FUNCTION_BLOCK UT_AuxiliaryInputMapping_Type_13_QuadratAnalog_Ret50perc (* Two quadrature mounted analog returns to centre position at 50% *)
  (* Standard: ISO 11783-6; Classification: AUX – ISO 11783-6; Function: All Inputs; Type: UT according to ISO 11783-6; Description: - Type 13 QuadratAnalog_Ret50perc Two quadrature mounted analog returns to centre position at 50% Applicable AUX-N only * maps to IW IW - Input WORD (16 Bit) *)
  (* Version 1.0, 2018-12-05, Jose Cabral *)
  (* Version 1.1, 2022-08-04, Franz Hoepfinger, HR Agrartechnik GmbH *)
  (* Version 1.2, 2023-01-05, Franz Hoepfinger, HR Agrartechnik GmbH *)
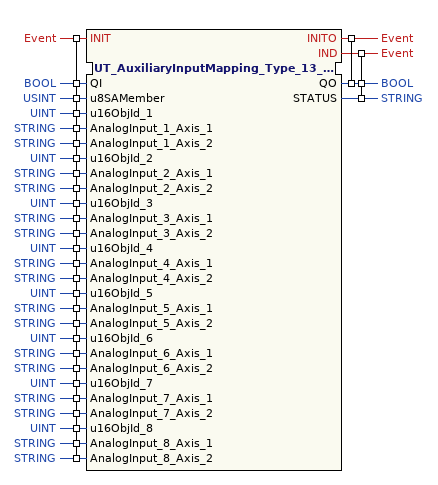
  EVENT_INPUT
    INIT WITH QI, u8SAMember, u16ObjId_1, AnalogInput_1_Axis_1, AnalogInput_1_Axis_2, u16ObjId_2, AnalogInput_2_Axis_1, AnalogInput_2_Axis_2, u16ObjId_3, AnalogInput_3_Axis_1, AnalogInput_3_Axis_2, u16ObjId_4, AnalogInput_4_Axis_1, AnalogInput_4_Axis_2, u16ObjId_5, AnalogInput_5_Axis_1, AnalogInput_5_Axis_2, u16ObjId_6, AnalogInput_6_Axis_1, AnalogInput_6_Axis_2, u16ObjId_7, AnalogInput_7_Axis_1, AnalogInput_7_Axis_2, u16ObjId_8, AnalogInput_8_Axis_1, AnalogInput_8_Axis_2; (* Service Initialization *)
  END_EVENT
  EVENT_OUTPUT
    INITO WITH QO; (* Initialization Confirm *)
    IND WITH QO, STATUS; (* Indication from Resource *)
  END_EVENT
  VAR_INPUT
    QI : BOOL; (* Event Input Qualifier *)
    u8SAMember : USINT := GLOBAL; (* Dummy !, set to GLOBAL if in doubt. OFF deactivates FB. *)
    u16ObjId_1 : UINT; (* Object ID of Input 1 *)
    AnalogInput_1_Axis_1 : STRING; (* Identifier for Input 1 Axis #1 *)
    AnalogInput_1_Axis_2 : STRING; (* Identifier for Input 1 Axis #2 *)
    u16ObjId_2 : UINT; (* Object ID of Input 2 *)
    AnalogInput_2_Axis_1 : STRING; (* Identifier for Input 2 Axis #1 *)
    AnalogInput_2_Axis_2 : STRING; (* Identifier for Input 2 Axis #2 *)
    u16ObjId_3 : UINT; (* Object ID of Input 3 *)
    AnalogInput_3_Axis_1 : STRING; (* Identifier for Input 3 Axis #1 *)
    AnalogInput_3_Axis_2 : STRING; (* Identifier for Input 3 Axis #2 *)
    u16ObjId_4 : UINT; (* Object ID of Input 4 *)
    AnalogInput_4_Axis_1 : STRING; (* Identifier for Input 4 Axis #1 *)
    AnalogInput_4_Axis_2 : STRING; (* Identifier for Input 4 Axis #2 *)
    u16ObjId_5 : UINT; (* Object ID of Input 5 *)
    AnalogInput_5_Axis_1 : STRING; (* Identifier for Input 5 Axis #1 *)
    AnalogInput_5_Axis_2 : STRING; (* Identifier for Input 5 Axis #2 *)
    u16ObjId_6 : UINT; (* Object ID of Input 6 *)
    AnalogInput_6_Axis_1 : STRING; (* Identifier for Input 6 Axis #1 *)
    AnalogInput_6_Axis_2 : STRING; (* Identifier for Input 6 Axis #2 *)
    u16ObjId_7 : UINT; (* Object ID of Input 7 *)
    AnalogInput_7_Axis_1 : STRING; (* Identifier for Input 7 Axis #1 *)
    AnalogInput_7_Axis_2 : STRING; (* Identifier for Input 7 Axis #2 *)
    u16ObjId_8 : UINT; (* Object ID of Input 8 *)
    AnalogInput_8_Axis_1 : STRING; (* Identifier for Input 8 Axis #1 *)
    AnalogInput_8_Axis_2 : STRING; (* Identifier for Input 8 Axis #2 *)
  END_VAR
  VAR_OUTPUT
    QO : BOOL; (* Event Output Qualifier *)
    STATUS : STRING; (* Service Status *)
  END_VAR
END_FUNCTION_BLOCK
